{attribute 'pack_mode' := '1'}
TYPE ST_ReadListData :
STRUCT
	stReadListReturnInfo	: ARRAY [1..gNodeIDCount] OF ST_UAReadListReturnInfo; // must be less than nMaxNodeIDsInList, nMaxNodeIDsInList = 10
	nIntVar1				: INT; 
	nIntVar2				: INT; 
	nIntVar3				: INT;
	nIntVar4				: INT;
	nIntVar5				: INT;
	nIntVar6				: INT;
	nIntVar7				: INT;
	nIntVar8				: INT;
	nIntVar9				: INT;
	nIntVar10				: INT;
END_STRUCT
END_TYPE

(* stored: Version 1.1.0.1, ProductVersion 3.1.4022.6
   DUT ST_ReadListData: Id {4e5213e3-ac25-4cd0-bcd3-8e0696bf7ac0} *)
